// TIA Portal V17 export
// export: Created 2025-04-11T04:54:25.0056241Z, ExportSetting WithDefaults, DisplayName Totally Integrated Automation Portal, DisplayVersion V17, DisplayName TIA Portal Openness, DisplayVersion V17, DisplayName TIA Portal Version Control Interface, DisplayVersion V17, DisplayName SINAMICS Startdrive Advanced, DisplayVersion V17, DisplayName SINAMICS Startdrive G130, G150, S120, S150, SINAMICS MV, S210, DisplayVersion V17, DisplayName SINAMICS Startdrive G110M, G120, G120C, G120D, G120P, G115D, DisplayVersion V17, DisplayName STEP 7 Professional, DisplayVersion V17, DisplayName STEP 7 Safety, DisplayVersion V17, DisplayName WinCC Advanced, DisplayVersion V17
TYPE "UDT_Ana_HMI"
// stored: IsFailsafeCompliant false
   STRUCT
      OUT_uiState : UInt;   // 状态字(0=初始状态,1=正常,2=高高报警,3=高报警,4=低报警,5=低低报警,6=传感器故障)
      OUT_EngValue : Real;   // 工程值
   END_STRUCT;
END_TYPE
